PROGRAM POU_AXIS
VAR
	fbExtruderAxis: MC_PowerStepper;
	fbHotendAxis: MC_Power;
END_VAR

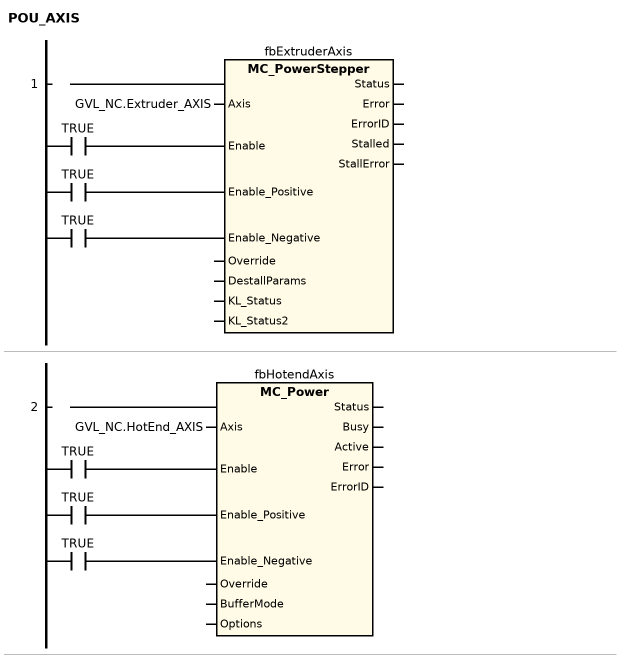
// NETWORK 1
fbExtruderAxis(
    Axis := GVL_NC.Extruder_AXIS,
    Enable := TRUE,
    Enable_Positive := TRUE,
    Enable_Negative := TRUE); // MC_PowerStepper

// NETWORK 2
fbHotendAxis(Axis := GVL_NC.HotEnd_AXIS, Enable := TRUE, Enable_Positive := TRUE, Enable_Negative := TRUE); // MC_Power

END_PROGRAM

(* stored: Version 1.1.0.1, ProductVersion 3.1.4024.2
   POU POU_AXIS: Id {53210104-c378-475f-82e5-3e9a7733a0d8}, SpecialFunc None *)
